PROGRAM Winder_data
VAR
	TP_0: TP;
	TP_1: TP;
	TP_2: TP;
	Power_lever_0: FB_Power_lever;
	Clutch_0: FB_Clutch;
	Mode_0: FB_Mode;
	Brake_0: FB_Brake;
	Standard_stuff_0: FB_Standard_stuff;
END_VAR

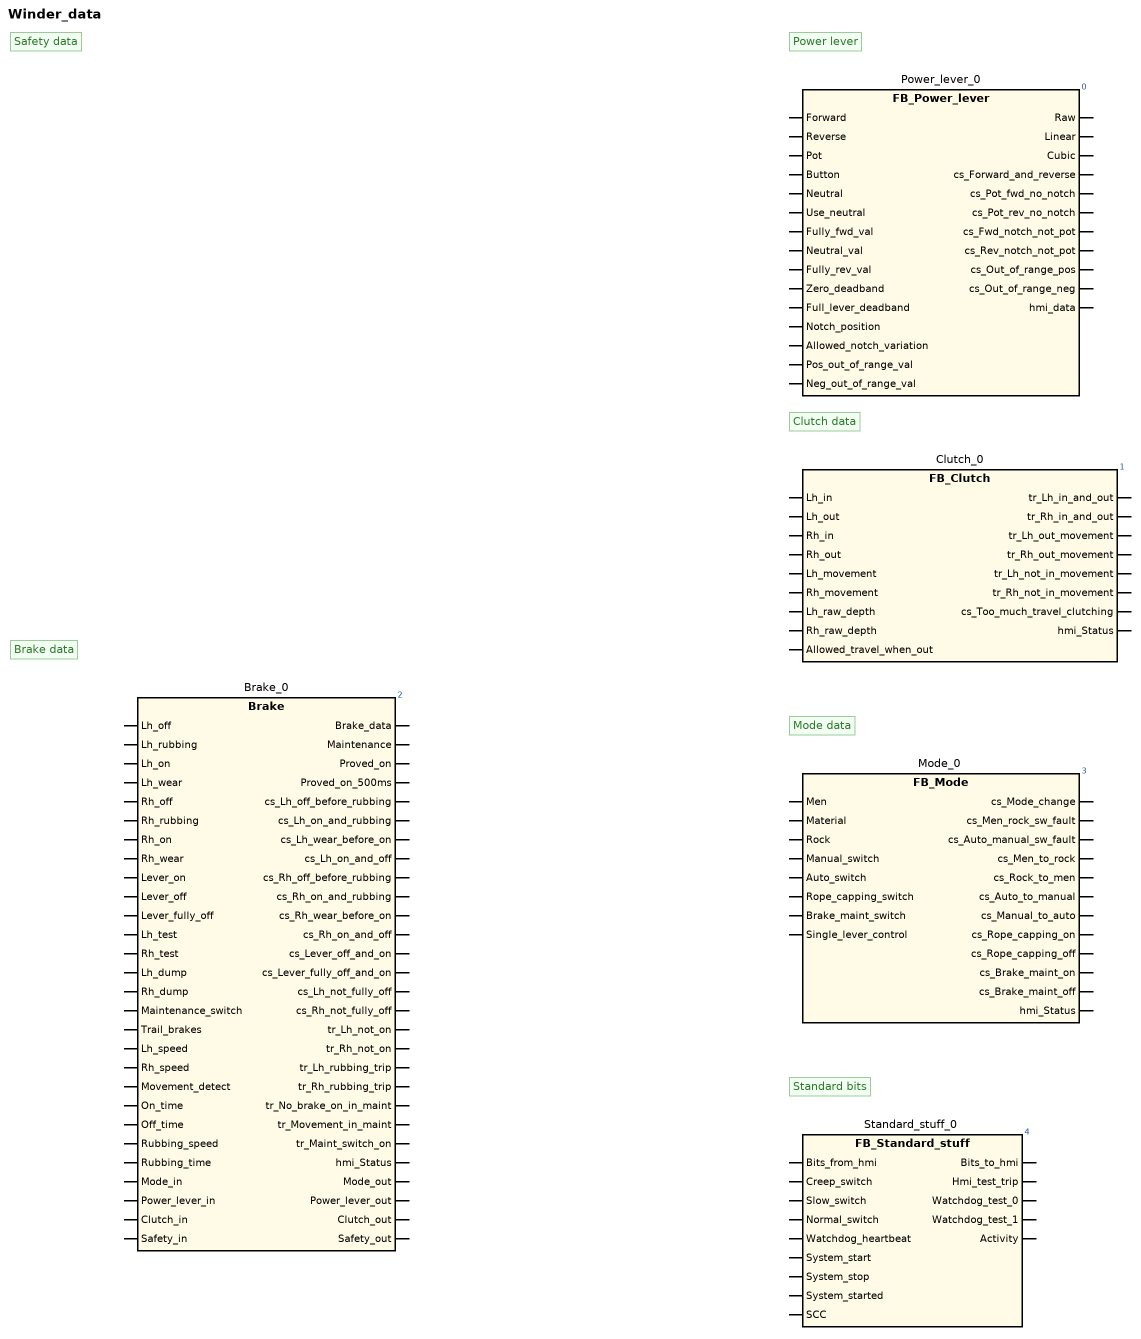
// Safety data
// Power lever
Power_lever_0(); // FB_Power_lever
// Clutch data
Clutch_0(); // FB_Clutch
// Brake data
Brake_0(); // Brake
// Mode data
Mode_0(); // FB_Mode
// Standard bits
Standard_stuff_0(); // FB_Standard_stuff

END_PROGRAM

(* stored: Version 1.1.0.1, ProductVersion 3.1.4024.0
   POU Winder_data: Id {adeaff29-a88d-4b52-a1fb-ee7f456997be}, SpecialFunc None *)
